{attribute 'pack_mode' := '2'}
TYPE ST_Out :
STRUCT

  bEnabled    : BIT; // Enabled: check if ControlLoop is closed and active
  bReferenced : BIT; // Axis homing bit
  bReady      : BIT; // enabled & NOT bError & no Axis Function requested
  bBusy       : BIT; // axis function requested or active
  bError      : BIT;
  bTimeout    : BIT; // for move cmds or switching drive on timeout
  bInTarget   : BIT; // ActPos = SetPos --> position check is done with configured window in NC
  bStandstill : BIT; // No Error and NOT moving

  byAxisFuncPara      : BYTE; // mirror for additional parameter for Axis Function; e.g. used for AxisIndex on GearIn
  uiAxisFunctionState : E_AXIS_STATE; // mirror the requested axis function; 
                                        // +  100 = function busy; 
                                        // + 1000 = function done; 
                                        // + 9000 = function error
  uiErrorId           : UDINT;

  rActPos             : LREAL;
  rActVelo            : LREAL;
  rPosDiff            : LREAL;

  // HAUD
  // 2023 04 05
  dwCoupleState       : DWORD;   // cyclic information about axis couple state

  NcAxisId            : UDINT;
END_STRUCT
END_TYPE

(* stored: Version 1.1.0.1, ProductVersion 3.1.4024.12
   DUT ST_Out: Id {b9820cfd-2679-41ef-bac5-055ca4628d56} *)
